INTERFACE I_Sensor

PROPERTY PUBLIC IsActive : BOOL
GET
END_GET
END_PROPERTY

END_INTERFACE

(* stored: Version 1.1.0.1, ProductVersion 3.1.4024.11
   Itf I_Sensor: Id {c1bf2c24-bb18-44a2-b237-4238fd24e21e}
   Property IsActive: Id {187bf708-8fe4-47a9-b22a-1a5672b32540}
   Get Get: Id {ae052df6-7d6d-4b41-982b-dbf1cc1e35a4} *)
